Yaskawa INFORM job: 12345678901234567.JBI

/JOB
//NAME 12345678901234567
//POS
///NPOS 0,0,0,1,0,0
///TOOL 0
///POSTYPE BASE
///RECTAN
///RCONF 0,0,0,0,0,0,0,0,0,0,0,0,0,0,0,0,0,0,0,0,0,0,0,0
P00000=0.000,0.000,0.000,0.0000,0.0000,0.0000
//INST
///DATE 2021/02/10 13:48
///ATTR SC,RW
///GROUP1 RB1
NOP
MOVJ P000 VJ=5.00
END
